{attribute 'qualified_only'}
{attribute 'strict'}
TYPE E_DataTypes :
(
	eBOOL	:= 0,
	eINT	:= 1,
	eReal	:= 2,
	eLreal	:= 3
	
);
END_TYPE

(* stored: Version 1.1.0.1, ProductVersion 3.1.4024.3
   DUT E_DataTypes: Id {77acbcf0-63a6-4a3c-a355-55a575060b64} *)
